FUNCTION_BLOCK BistableCylinder EXTENDS BaseCylinder
VAR_INPUT	
END_VAR
VAR_OUTPUT
END_VAR
VAR	
	//Hardware
	DO_Retract AT %Q* : BOOL;
END_VAR

METHOD METH_Extend : BOOL
DO_Extend := TRUE;
DO_Retract := FALSE;
END_METHOD

METHOD METH_Retract : BOOL
DO_Extend := FALSE;
DO_Retract := TRUE;
END_METHOD

END_FUNCTION_BLOCK

(* stored: Version 1.1.0.1
   POU BistableCylinder: Id {1b0a2d23-6a30-4858-9d0b-91c9b4437b43}, SpecialFunc None
   Method METH_Extend: Id {082aed2c-388d-46f9-9e5e-63ba4724abab}
   Method METH_Retract: Id {673313ca-267e-409b-8754-ad44b648399c} *)
